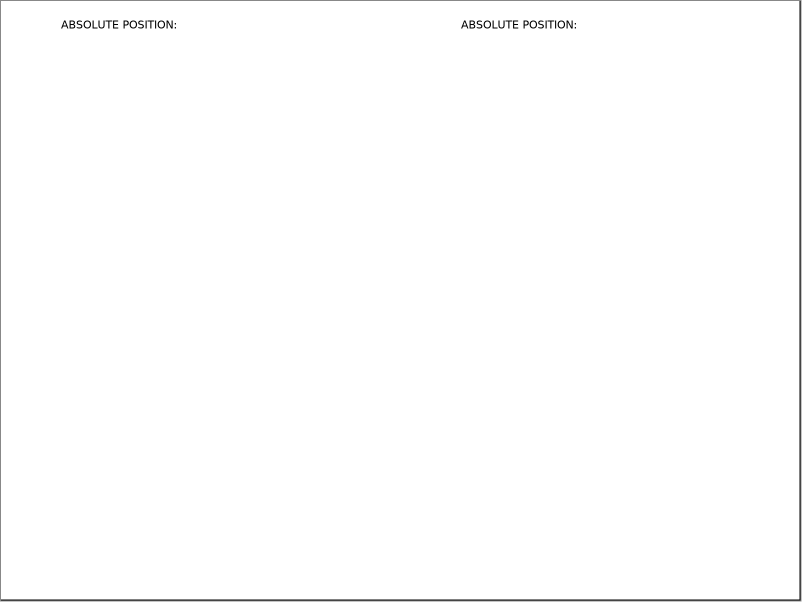
VISUALIZATION F19_Touch_Probe  // 802x602
    Rectangle (0,0 800x600)
    Label (10,10 170x30), "ABSOLUTE POSITION:"
    Label (410,10 170x30), "ABSOLUTE POSITION:"
END_VISUALIZATION

(* stored: Version 1.1.0.1, ProductVersion 3.1.4022.7
   Visu F19_Touch_Probe: Id {60dda6c2-b5e3-46ff-92fc-dc268987d202} *)
